FUNCTION_BLOCK FB_CellCheckPart_Test EXTENDS TcUnit.FB_TestSuite
VAR
END_VAR

CheckPartGood();
CheckPartBadBarcode();

METHOD PRIVATE CheckPartBadBarcode
VAR
	fbCell		: ADO_Demo_PLC.FB_Cell;
	MockStatus	: ADO_Demo_PLC.ST_PartStatus;
	Expected	: BOOL := FALSE;
	Result		: BOOL;
END_VAR
MockStatus.bBarcodeStatus := FALSE;
MockStatus.bCapperStatus := TRUE;
MockStatus.bFillerStatus := TRUE;
MockStatus.bWeightStatus := TRUE;

Result := fbCell.CheckPart(MockStatus);

AssertEquals(Expected := Expected,
             Actual := Result,
             Message := 'part check mismatch');

TEST_FINISHED();
END_METHOD

METHOD PRIVATE CheckPartGood
VAR
	fbCell		: ADO_Demo_PLC.FB_Cell;
	MockStatus	: ADO_Demo_PLC.ST_PartStatus;
	Expected	: BOOL := TRUE;
	Result		: BOOL;
END_VAR
MockStatus.bBarcodeStatus := TRUE;
MockStatus.bCapperStatus := TRUE;
MockStatus.bFillerStatus := TRUE;
MockStatus.bWeightStatus := TRUE;

Result := fbCell.CheckPart(MockStatus);

AssertEquals(Expected := Expected,
             Actual := Result,
             Message := 'part check mismatch');

TEST_FINISHED();
END_METHOD

END_FUNCTION_BLOCK

(* stored: Version 1.1.0.1, ProductVersion 3.1.4024.12
   POU FB_CellCheckPart_Test: Id {914beea1-202e-4b67-bb05-8582061c407a}, SpecialFunc None
   Method CheckPartBadBarcode: Id {e93e06dc-8d24-4945-af9a-ab9e2dbce2fd}
   Method CheckPartGood: Id {200cbed5-bc77-47d7-ad2e-8ab6e19818c3} *)
